// TwinCAT 3 PLC project mobject_packml
// Title: mobject-packml
// Company: mobject.io
// Author: mobject dev team
// ProjectVersion: 0.1.0
// ProgramVersion: 3.1.4023.0
// libraries:
//   Tc2_System, * (Beckhoff Automation GmbH)
// project tree:
//   PackMl Mode/ I_PackML_Mode.TcIO, PackML_Mode.TcPOU
//   _Internal/DUT/ PackML_State.TcDUT
//   _Internal/Interface/ I_PackML_AbortedCommands.TcIO, I_PackML_AbortingCommands.TcIO, I_PackML_ClearningCommands.TcIO, I_PackML_CompleteCommands.TcIO, I_PackML_CompletingCommands.TcIO, I_PackML_ExecuteCommands.TcIO, I_PackML_HeldCommands.TcIO, I_PackML_HoldingCommands.TcIO, I_PackML_IdleCommands.TcIO, I_PackML_ResettingCommands.TcIO, I_PackML_StartingCommands.TcIO, I_PackML_StoppedCommands.TcIO, I_PackML_StoppingCommands.TcIO, I_PackML_SuspendedCommands.TcIO, I_PackML_SuspendingCommands.TcIO, I_PackML_UnholdingCommands.TcIO, I_PackML_UnsuspendingCommands.TcIO
//   _Internal/StateMachine/ PackMLStateMachine.TcPOU

// ---- _Internal/DUT/PackML_State.TcDUT
{attribute 'qualified_only'}
{attribute 'strict'}
TYPE PackML_State :
(
	UNDEFINED := 0,
    CLEARING := 1,
    STOPPED := 2,
    STARTING := 3,
    IDLE := 4,
    SUSPENDED := 5,
	EXECUTE := 6,
    STOPPING := 7,
    ABORTING := 8,
    ABORTED := 9,
    HOLDING := 10,
    HELD := 11,
    UNHOLDING := 12,
    SUSPENDING := 13,
    UNSUSPENDING := 14,
    RESETTING := 15,
    COMPLETING := 16,
    COMPLETE := 17
);
END_TYPE

// ---- PackMl Mode/I_PackML_Mode.TcIO
INTERFACE I_PackML_Mode

METHOD PUBLIC Abort
VAR_INPUT
END_VAR
END_METHOD

METHOD PUBLIC Clear
VAR_INPUT
END_VAR
END_METHOD

PROPERTY PUBLIC CurrentState : PackML_State
GET
END_GET
END_PROPERTY

METHOD PUBLIC CyclicCall
VAR_INPUT
END_VAR
END_METHOD

METHOD PUBLIC Hold
VAR_INPUT
END_VAR
END_METHOD

PROPERTY PUBLIC IsAborted : bool
GET
END_GET
END_PROPERTY

PROPERTY PUBLIC IsAborting : bool
GET
END_GET
END_PROPERTY

PROPERTY PUBLIC IsClearing : bool
GET
END_GET
END_PROPERTY

PROPERTY PUBLIC IsComplete : bool
GET
END_GET
END_PROPERTY

PROPERTY PUBLIC IsCompleting : bool
GET
END_GET
END_PROPERTY

PROPERTY PUBLIC IsExecuting : bool
GET
END_GET
END_PROPERTY

PROPERTY PUBLIC IsHeld : bool
GET
END_GET
END_PROPERTY

PROPERTY PUBLIC IsHolding : bool
GET
END_GET
END_PROPERTY

PROPERTY PUBLIC IsIdle : BOOL
GET
END_GET
END_PROPERTY

METHOD PUBLIC IsModeTransitionAllowed : BOOL
VAR_INPUT
	
END_VAR
END_METHOD

PROPERTY PUBLIC IsResetting : bool
GET
END_GET
END_PROPERTY

PROPERTY PUBLIC IsStarting : bool
GET
END_GET
END_PROPERTY

PROPERTY PUBLIC IsStopped : BOOL
GET
END_GET
END_PROPERTY

PROPERTY PUBLIC IsStopping : bool
GET
END_GET
END_PROPERTY

PROPERTY PUBLIC IsSuspended : bool
GET
END_GET
END_PROPERTY

PROPERTY PUBLIC IsSuspending : bool
GET
END_GET
END_PROPERTY

PROPERTY PUBLIC IsUnholding : bool
GET
END_GET
END_PROPERTY

PROPERTY PUBLIC IsUnsuspending : bool
GET
END_GET
END_PROPERTY

METHOD PUBLIC Reset
VAR_INPUT
END_VAR
END_METHOD

METHOD PUBLIC Start
VAR_INPUT
END_VAR
END_METHOD

METHOD PUBLIC Stop
VAR_INPUT
END_VAR
END_METHOD

METHOD PUBLIC Suspend
VAR_INPUT
END_VAR
END_METHOD

METHOD PUBLIC Unhold
VAR_INPUT
END_VAR
END_METHOD

METHOD PUBLIC Unsuspend
VAR_INPUT
END_VAR
END_METHOD

END_INTERFACE

// ---- _Internal/Interface/I_PackML_AbortedCommands.TcIO
INTERFACE I_PackML_AbortedCommands

METHOD PUBLIC Clear
VAR_INPUT
END_VAR
END_METHOD

END_INTERFACE

// ---- _Internal/Interface/I_PackML_AbortingCommands.TcIO
INTERFACE I_PackML_AbortingCommands

METHOD StateComplete
VAR_INPUT
END_VAR
END_METHOD

END_INTERFACE

// ---- _Internal/Interface/I_PackML_ClearningCommands.TcIO
INTERFACE I_PackML_ClearningCommands

METHOD PUBLIC Abort
VAR_INPUT
END_VAR
END_METHOD

METHOD StateComplete
VAR_INPUT
END_VAR
END_METHOD

END_INTERFACE

// ---- _Internal/Interface/I_PackML_CompleteCommands.TcIO
INTERFACE I_PackML_CompleteCommands

METHOD PUBLIC Abort
VAR_INPUT
END_VAR
END_METHOD

METHOD PUBLIC Reset
VAR_INPUT
END_VAR
END_METHOD

METHOD PUBLIC Stop
VAR_INPUT
END_VAR
END_METHOD

END_INTERFACE

// ---- _Internal/Interface/I_PackML_CompletingCommands.TcIO
INTERFACE I_PackML_CompletingCommands

METHOD PUBLIC Abort
VAR_INPUT
END_VAR
END_METHOD

METHOD StateComplete
VAR_INPUT
END_VAR
END_METHOD

METHOD PUBLIC Stop
VAR_INPUT
END_VAR
END_METHOD

END_INTERFACE

// ---- _Internal/Interface/I_PackML_ExecuteCommands.TcIO
INTERFACE I_PackML_ExecuteCommands

METHOD PUBLIC Abort
VAR_INPUT
END_VAR
END_METHOD

METHOD PUBLIC Hold
VAR_INPUT
END_VAR
END_METHOD

METHOD StateComplete
VAR_INPUT
END_VAR
END_METHOD

METHOD PUBLIC Stop
VAR_INPUT
END_VAR
END_METHOD

METHOD PUBLIC Suspend
VAR_INPUT
END_VAR
END_METHOD

END_INTERFACE

// ---- _Internal/Interface/I_PackML_HeldCommands.TcIO
INTERFACE I_PackML_HeldCommands

METHOD PUBLIC Abort
VAR_INPUT
END_VAR
END_METHOD

METHOD PUBLIC Stop
VAR_INPUT
END_VAR
END_METHOD

METHOD PUBLIC Unhold
VAR_INPUT
END_VAR
END_METHOD

END_INTERFACE

// ---- _Internal/Interface/I_PackML_HoldingCommands.TcIO
INTERFACE I_PackML_HoldingCommands

METHOD PUBLIC Abort
VAR_INPUT
END_VAR
END_METHOD

METHOD StateComplete
VAR_INPUT
END_VAR
END_METHOD

METHOD PUBLIC Stop
VAR_INPUT
END_VAR
END_METHOD

END_INTERFACE

// ---- _Internal/Interface/I_PackML_IdleCommands.TcIO
INTERFACE I_PackML_IdleCommands

METHOD PUBLIC Abort
VAR_INPUT
END_VAR
END_METHOD

METHOD PUBLIC Start
VAR_INPUT
END_VAR
END_METHOD

METHOD PUBLIC Stop
VAR_INPUT
END_VAR
END_METHOD

END_INTERFACE

// ---- _Internal/Interface/I_PackML_ResettingCommands.TcIO
INTERFACE I_PackML_ResettingCommands

METHOD PUBLIC Abort
VAR_INPUT
END_VAR
END_METHOD

METHOD StateComplete
VAR_INPUT
END_VAR
END_METHOD

METHOD PUBLIC Stop
VAR_INPUT
END_VAR
END_METHOD

END_INTERFACE

// ---- _Internal/Interface/I_PackML_StartingCommands.TcIO
INTERFACE I_PackML_StartingCommands

METHOD PUBLIC Abort
VAR_INPUT
END_VAR
END_METHOD

METHOD StateComplete
VAR_INPUT
END_VAR
END_METHOD

METHOD PUBLIC Stop
VAR_INPUT
END_VAR
END_METHOD

END_INTERFACE

// ---- _Internal/Interface/I_PackML_StoppedCommands.TcIO
INTERFACE I_PackML_StoppedCommands

METHOD PUBLIC Abort
VAR_INPUT
END_VAR
END_METHOD

METHOD PUBLIC Reset
VAR_INPUT
END_VAR
END_METHOD

END_INTERFACE

// ---- _Internal/Interface/I_PackML_StoppingCommands.TcIO
INTERFACE I_PackML_StoppingCommands

METHOD PUBLIC Abort
VAR_INPUT
END_VAR
END_METHOD

METHOD StateComplete
VAR_INPUT
END_VAR
END_METHOD

END_INTERFACE

// ---- _Internal/Interface/I_PackML_SuspendedCommands.TcIO
INTERFACE I_PackML_SuspendedCommands

METHOD PUBLIC Abort
VAR_INPUT
END_VAR
END_METHOD

METHOD PUBLIC Stop
VAR_INPUT
END_VAR
END_METHOD

METHOD PUBLIC Unsuspend
VAR_INPUT
END_VAR
END_METHOD

END_INTERFACE

// ---- _Internal/Interface/I_PackML_SuspendingCommands.TcIO
INTERFACE I_PackML_SuspendingCommands

METHOD PUBLIC Abort
VAR_INPUT
END_VAR
END_METHOD

METHOD StateComplete
VAR_INPUT
END_VAR
END_METHOD

METHOD PUBLIC Stop
VAR_INPUT
END_VAR
END_METHOD

END_INTERFACE

// ---- _Internal/Interface/I_PackML_UnholdingCommands.TcIO
INTERFACE I_PackML_UnholdingCommands

METHOD PUBLIC Abort
VAR_INPUT
END_VAR
END_METHOD

METHOD StateComplete
VAR_INPUT
END_VAR
END_METHOD

METHOD PUBLIC Stop
VAR_INPUT
END_VAR
END_METHOD

END_INTERFACE

// ---- _Internal/Interface/I_PackML_UnsuspendingCommands.TcIO
INTERFACE I_PackML_UnsuspendingCommands

METHOD PUBLIC Abort
VAR_INPUT
END_VAR
END_METHOD

METHOD StateComplete
VAR_INPUT
END_VAR
END_METHOD

METHOD PUBLIC Stop
VAR_INPUT
END_VAR
END_METHOD

END_INTERFACE

// ---- PackMl Mode/PackML_Mode.TcPOU
{attribute 'linkalways'} 
{attribute 'no_explicit_call' := 'This FB is a CLASS and must be accessed using methods or properties'}
{attribute 'enable_dynamic_creation'}
FUNCTION_BLOCK PackML_Mode IMPLEMENTS I_PackML_Mode
VAR
	packMLStateMachine : PackMLStateMachine;
END_VAR

METHOD PUBLIC Abort
VAR_INPUT
END_VAR
packMLStateMachine.Abort();
END_METHOD

METHOD PROTECTED Aborted
VAR_INPUT
	Commands : I_PackML_AbortedCommands;
END_VAR
END_METHOD

METHOD PROTECTED Aborting
VAR_INPUT
	Commands : I_PackML_AbortingCommands;
END_VAR
Commands.StateComplete();
END_METHOD

METHOD PUBLIC Clear
VAR_INPUT
END_VAR
packMLStateMachine.Clear();
END_METHOD

METHOD PROTECTED Clearing
VAR_INPUT
	Commands : I_PackML_ClearningCommands;
END_VAR
Commands.StateComplete();
END_METHOD

METHOD PROTECTED Complete
VAR_INPUT
	Commands : I_PackML_CompleteCommands;
END_VAR
END_METHOD

METHOD PROTECTED Completing
VAR_INPUT
	Commands : I_PackML_CompletingCommands;
END_VAR
Commands.StateComplete();
END_METHOD

PROPERTY PUBLIC CurrentState : PackML_State
GET
CurrentState := packMLStateMachine.CurrentState;
END_GET
END_PROPERTY

METHOD PUBLIC CyclicCall
VAR_INPUT
END_VAR
IF packMLStateMachine.IsIdle THEN 
	Idle(packMLStateMachine);
END_IF

IF packMLStateMachine.IsStarting THEN
	Starting(packMLStateMachine);
END_IF

IF packMLStateMachine.IsExecuting THEN
	Execute(packMLStateMachine);
END_IF

IF packMLStateMachine.IsCompleting THEN
	Completing(packMLStateMachine);
END_IF

IF packMLStateMachine.IsComplete THEN
	Complete(packMLStateMachine);
END_IF

IF packMLStateMachine.IsStopping THEN
	Stopping(packMLStateMachine);
END_IF

IF packMLStateMachine.IsStopped THEN
	Stopped(packMLStateMachine);
END_IF

IF packMLStateMachine.IsResetting THEN
	Resetting(packMLStateMachine);
END_IF

IF packMLStateMachine.IsHolding THEN
	Holding(packMLStateMachine);
END_IF

IF packMLStateMachine.IsHeld THEN
	Held(packMLStateMachine);
END_IF

IF packMLStateMachine.IsUnholding THEN
	Unholding(packMLStateMachine);
END_IF

IF packMLStateMachine.IsSuspending THEN
	Suspending(packMLStateMachine);
END_IF

IF packMLStateMachine.IsSuspended THEN
	Suspended(packMLStateMachine);
END_IF

IF packMLStateMachine.IsUnsuspending THEN
	Unsuspending(packMLStateMachine);
END_IF

IF packMLStateMachine.IsClearing THEN
	Clearing(packMLStateMachine);
END_IF

IF packMLStateMachine.IsAborted THEN
	Aborted(packMLStateMachine);
END_IF

IF packMLStateMachine.IsAborting THEN
	Aborting(packMLStateMachine);
END_IF
END_METHOD

METHOD PROTECTED Execute
VAR_INPUT
	Commands : I_PackML_ExecuteCommands;
END_VAR
Commands.StateComplete();
END_METHOD

METHOD PROTECTED Held
VAR_INPUT
	Commands : I_PackML_HeldCommands;
END_VAR
END_METHOD

METHOD PUBLIC Hold
VAR_INPUT
END_VAR
packMLStateMachine.Hold();
END_METHOD

METHOD PROTECTED Holding
VAR_INPUT
	Commands : I_PackML_HoldingCommands;
END_VAR
Commands.StateComplete();
END_METHOD

METHOD PROTECTED Idle
VAR_INPUT
	Commands : I_PackML_IdleCommands;
END_VAR
END_METHOD

PROPERTY PUBLIC IsAborted : bool
GET
IsAborted := packMLStateMachine.IsAborted;
END_GET
END_PROPERTY

PROPERTY PUBLIC IsAborting : bool
GET
IsAborting := packMLStateMachine.IsAborting;
END_GET
END_PROPERTY

PROPERTY PUBLIC IsClearing : bool
GET
IsClearing := packMLStateMachine.IsClearing;
END_GET
END_PROPERTY

PROPERTY PUBLIC IsComplete : bool
GET
IsComplete := packMLStateMachine.IsComplete;
END_GET
END_PROPERTY

PROPERTY PUBLIC IsCompleting : bool
GET
IsCompleting := packMLStateMachine.IsCompleting;
END_GET
END_PROPERTY

PROPERTY PUBLIC IsExecuting : bool
GET
IsExecuting := packMLStateMachine.IsExecuting;
END_GET
END_PROPERTY

PROPERTY PUBLIC IsHeld : bool
GET
IsHeld := packMLStateMachine.IsHeld;
END_GET
END_PROPERTY

PROPERTY PUBLIC IsHolding : bool
GET
IsHolding := packMLStateMachine.IsHolding;
END_GET
END_PROPERTY

PROPERTY PUBLIC IsIdle : BOOL
GET
isIdle := packMLStateMachine.isIdle;
END_GET
END_PROPERTY

METHOD PUBLIC IsModeTransitionAllowed : BOOL
VAR_INPUT
END_VAR
IsModeTransitionAllowedCheck(packMLStateMachine.CurrentState);
END_METHOD

METHOD PROTECTED IsModeTransitionAllowedCheck : BOOL
VAR_INPUT
	CurrentState : PackML_State;
END_VAR
IsModeTransitionAllowedCheck := true;
END_METHOD

PROPERTY PUBLIC IsResetting : bool
GET
IsResetting := packMLStateMachine.IsResetting;
END_GET
END_PROPERTY

PROPERTY PUBLIC IsStarting : bool
GET
IsStarting := packMLStateMachine.IsStarting;
END_GET
END_PROPERTY

PROPERTY PUBLIC IsStopped : BOOL
GET
isStopped := packMLStateMachine.isStopped;
END_GET
END_PROPERTY

PROPERTY PUBLIC IsStopping : bool
GET
IsStopping := packMLStateMachine.IsStopping;
END_GET
END_PROPERTY

PROPERTY PUBLIC IsSuspended : bool
GET
IsSuspended := packMLStateMachine.IsSuspended;
END_GET
END_PROPERTY

PROPERTY PUBLIC IsSuspending : bool
GET
IsSuspending := packMLStateMachine.IsSuspending;
END_GET
END_PROPERTY

PROPERTY PUBLIC IsUnholding : bool
GET
IsUnholding := packMLStateMachine.IsUnholding;
END_GET
END_PROPERTY

PROPERTY PUBLIC IsUnsuspending : bool
GET
IsUnsuspending := packMLStateMachine.IsUnsuspending;
END_GET
END_PROPERTY

METHOD PUBLIC Reset
VAR_INPUT
END_VAR
packMLStateMachine.Reset();
END_METHOD

METHOD PROTECTED Resetting
VAR_INPUT
	Commands : I_PackML_ResettingCommands;
END_VAR
Commands.StateComplete();
END_METHOD

METHOD PUBLIC Start
VAR_INPUT
END_VAR
packMLStateMachine.Start();
END_METHOD

METHOD PROTECTED Starting
VAR_INPUT
	Commands : I_PackML_StartingCommands;
END_VAR
Commands.StateComplete();
END_METHOD

METHOD PUBLIC Stop
VAR_INPUT
END_VAR
packMLStateMachine.Stop();
END_METHOD

METHOD PROTECTED Stopped
VAR_INPUT
	Commands : I_PackML_StoppedCommands;
END_VAR
END_METHOD

METHOD PROTECTED Stopping
VAR_INPUT
	Commands : I_PackML_StoppingCommands;
END_VAR
Commands.StateComplete();
END_METHOD

METHOD PUBLIC Suspend
VAR_INPUT
END_VAR
packMLStateMachine.Suspend();
END_METHOD

METHOD PROTECTED Suspended
VAR_INPUT
	Commands : I_PackML_SuspendedCommands;
END_VAR
END_METHOD

METHOD PROTECTED Suspending
VAR_INPUT
	Commands : I_PackML_SuspendingCommands;
END_VAR
Commands.StateComplete();
END_METHOD

METHOD PUBLIC Unhold
VAR_INPUT
END_VAR
packMLStateMachine.Unhold();
END_METHOD

METHOD PROTECTED Unholding
VAR_INPUT
	Commands : I_PackML_UnholdingCommands;
END_VAR
Commands.StateComplete();
END_METHOD

METHOD PUBLIC Unsuspend
VAR_INPUT
END_VAR
packMLStateMachine.Unsuspend();
END_METHOD

METHOD PROTECTED Unsuspending
VAR_INPUT
	Commands : I_PackML_UnsuspendingCommands;
END_VAR
Commands.StateComplete();
END_METHOD

END_FUNCTION_BLOCK

// ---- _Internal/StateMachine/PackMLStateMachine.TcPOU
{attribute 'linkalways'} 
{attribute 'no_explicit_call' := 'This FB is a CLASS and must be accessed using methods or properties'}
{attribute 'enable_dynamic_creation'}
FUNCTION_BLOCK PackMLStateMachine IMPLEMENTS I_PackML_AbortingCommands,I_PackML_ClearningCommands,I_PackML_HeldCommands, I_PackML_CompletingCommands,I_PackML_ExecuteCommands,I_PackML_AbortedCommands,I_PackML_CompleteCommands,I_PackML_HoldingCommands,I_PackML_UnsuspendingCommands,I_PackML_UnholdingCommands,I_PackML_SuspendingCommands,I_PackML_SuspendedCommands,I_PackML_IdleCommands,I_PackML_ResettingCommands,I_PackML_StartingCommands,I_PackML_StoppedCommands,I_PackML_StoppingCommands
VAR
	state : PackML_State := PackML_State.IDLE;
END_VAR

METHOD PUBLIC Abort
VAR_INPUT
END_VAR
IF IsAborting OR IsAborted THEN
	RETURN;
END_IF

state := PackML_State.ABORTING;
END_METHOD

METHOD PUBLIC Clear
VAR_INPUT
END_VAR
IF IsAborted THEN 
	state := PackML_State.CLEARING;
END_IF
END_METHOD

PROPERTY PUBLIC CurrentState : PackML_State
GET
CurrentState := state;
END_GET
END_PROPERTY

METHOD PUBLIC Hold
VAR_INPUT
END_VAR
IF IsExecuting THEN 
	state := PackML_State.HOLDING;
END_IF
END_METHOD

PROPERTY PUBLIC IsAborted : bool
GET
IsAborted := (state = PackML_State.ABORTED);
END_GET
END_PROPERTY

PROPERTY PUBLIC IsAborting : bool
GET
IsAborting := (state = PackML_State.ABORTING);
END_GET
END_PROPERTY

PROPERTY PUBLIC IsClearing : bool
GET
IsClearing := (state = PackML_State.CLEARING);
END_GET
END_PROPERTY

PROPERTY PUBLIC IsComplete : bool
GET
IsComplete := (state = PackML_State.COMPLETE);
END_GET
END_PROPERTY

PROPERTY PUBLIC IsCompleting : bool
GET
IsCompleting := (state = PackML_State.COMPLETING);
END_GET
END_PROPERTY

PROPERTY PUBLIC IsExecuting : bool
GET
IsExecuting := (state = PackML_State.EXECUTE);
END_GET
END_PROPERTY

PROPERTY PUBLIC IsHeld : bool
GET
IsHeld := (state = PackML_State.HELD);
END_GET
END_PROPERTY

PROPERTY PUBLIC IsHolding : bool
GET
IsHolding := (state = PackML_State.HOLDING);
END_GET
END_PROPERTY

PROPERTY PUBLIC IsIdle : BOOL
GET
isIdle := (state = PackML_State.IDLE);
END_GET
END_PROPERTY

PROPERTY PUBLIC IsResetting : bool
GET
IsResetting := (state = PackML_State.RESETTING);
END_GET
END_PROPERTY

PROPERTY PUBLIC IsStarting : bool
GET
IsStarting := (state = PackML_State.STARTING);
END_GET
END_PROPERTY

PROPERTY PUBLIC IsStopped : BOOL
GET
isStopped := (state = PackML_State.STOPPED);
END_GET
END_PROPERTY

PROPERTY PUBLIC IsStopping : bool
GET
IsStopping := (state = PackML_State.STOPPING);
END_GET
END_PROPERTY

PROPERTY PUBLIC IsSuspended : bool
GET
IsSuspended := (state = PackML_State.SUSPENDED);
END_GET
END_PROPERTY

PROPERTY PUBLIC IsSuspending : bool
GET
IsSuspending := (state = PackML_State.SUSPENDING);
END_GET
END_PROPERTY

PROPERTY PUBLIC IsUnholding : bool
GET
IsUnholding := (state = PackML_State.UNHOLDING);
END_GET
END_PROPERTY

PROPERTY PUBLIC IsUnsuspending : bool
GET
IsUnsuspending := (state = PackML_State.UNSUSPENDING);
END_GET
END_PROPERTY

METHOD PUBLIC Reset
VAR_INPUT
END_VAR
IF IsStopped OR IsComplete THEN 
	state := PackML_State.RESETTING;
END_IF
END_METHOD

METHOD PUBLIC Start
VAR_INPUT
END_VAR
IF IsIdle THEN 
	state := PackML_State.STARTING;
END_IF
END_METHOD

METHOD StateComplete
VAR_INPUT
END_VAR
CASE state OF 
	
	PackML_State.IDLE : RETURN;
	PackML_State.STARTING : state := PackML_State.EXECUTE;
	PackML_State.EXECUTE : state := PackML_State.COMPLETING;
	PackML_State.COMPLETING : state := PackML_State.COMPLETE;
	PackML_State.COMPLETE : RETURN;
	PackML_State.STOPPING : state := PackML_State.STOPPED;
	PackML_State.STOPPED : RETURN;
	PackML_State.RESETTING : state := PackML_State.IDLE;
	PackML_State.HOLDING : state := PackML_State.HELD;
	PackML_State.HELD : RETURN;
	PackML_State.UNHOLDING : state := PackML_State.EXECUTE;
	PackML_State.SUSPENDING : state := PackML_State.SUSPENDED;
	PackML_State.SUSPENDED : RETURN;
	PackML_State.UNSUSPENDING : state := PackML_State.EXECUTE;
	PackML_State.CLEARING : state := PackML_State.STOPPED;
	PackML_State.ABORTED : RETURN;
	PackML_State.ABORTING : state := PackML_State.ABORTED;
	
END_CASE
END_METHOD

METHOD PUBLIC Stop
VAR_INPUT
END_VAR
CASE state OF
	PackML_State.STOPPED: RETURN;
	PackML_State.STOPPING: RETURN;
	PackML_State.CLEARING: RETURN;
	PackML_State.ABORTED: RETURN;
	PackML_State.ABORTING: RETURN;
END_CASE

state := PackML_State.STOPPING;
END_METHOD

METHOD PUBLIC Suspend
VAR_INPUT
END_VAR
IF IsExecuting THEN 
	state := PackML_State.SUSPENDING;
END_IF
END_METHOD

METHOD PUBLIC Unhold
VAR_INPUT
END_VAR
IF IsHeld THEN 
	state := PackML_State.UNHOLDING;
END_IF
END_METHOD

METHOD PUBLIC Unsuspend
VAR_INPUT
END_VAR
IF IsSuspended THEN 
	state := PackML_State.UNSUSPENDING;
END_IF
END_METHOD

END_FUNCTION_BLOCK
